(* Logix 5000 project; controller cal1632 1756-L62 rev 16.20; software revision 16.05; part 31 of 61 *)
(* tags used below, declared in another part *)
   FAULT : BOOL;
   p01r09_pb_global_reset : BOOL;
   p21_ai_splice_platen_temp : REAL;
   p21_ao_splice_platen_temp_cv : REAL;
   p21_di_close_exit_clamp : BOOL;
   p21_di_close_inlet_clamp : BOOL;
   p21_di_open_splice_platen : BOOL;
   p21_di_platen_hi_temp_ok : BOOL;
   p21_di_platen_not_closed : BOOL;
   p21_di_splice_2_hand_close : BOOL;
   p21_di_tc_bo : BOOL;
   p21_dint_to_hmi : DINT[16];
   p21_do_close_exit_clamp_sv : BOOL;
   p21_do_close_inlet_clamp_sv : BOOL;
   p21_do_close_platen_sv : BOOL;
   p21_do_enable_platen_heater : BOOL;
   p21_real_to_hmi : REAL[112];
   p21_splice_press_temp_out : SYS_SCP;
   p21_splice_temp_in_max : REAL;
   p21_splice_temp_in_min : REAL;
   p21_splice_temp_out_max : REAL;
   p21_splice_temp_out_min : REAL;
   P21r01 : routine;
   p21r02 : routine;
   p21r02_fault_exists : BOOL;
   p21r02_timer_fault : TIMER[4];
   p21r02_timer_warning : TIMER[4];
   p21r02_unack_fault : BOOL;
   p21r02_unack_warning : BOOL;
   p21r02_warning_exists : BOOL;
   p21r03 : routine;
   p21r03_timer_fault : TIMER[4];
   p21r03_timer_warning : TIMER[4];
   p21r04 : routine;
   p21r04_timer_fault : TIMER[4];
   p21r04_timer_warning : TIMER[4];
   p21r05 : routine;
   p21r05_timer_fault : TIMER[4];
   p21r05_timer_warning : TIMER[4];
   p21r06 : routine;
   p21r06_timer_fault : TIMER[4];
   p21r06_timer_warning : TIMER[4];
   p21r07 : routine;
   p21r08 : routine;
   p21r09 : routine;
   p21r10 : routine;
   p21r10_remaining_cure_time_sec : REAL;
   p21r10_status : DINT;
   p21r16 : routine;
   p21r16_pid_temp_cv : REAL;
   p21r16_request_heat : BOOL;

PROGRAM P21_Splice_Press   (* main routine R01_Main *)

ROUTINE R01_Main   (* ladder *)
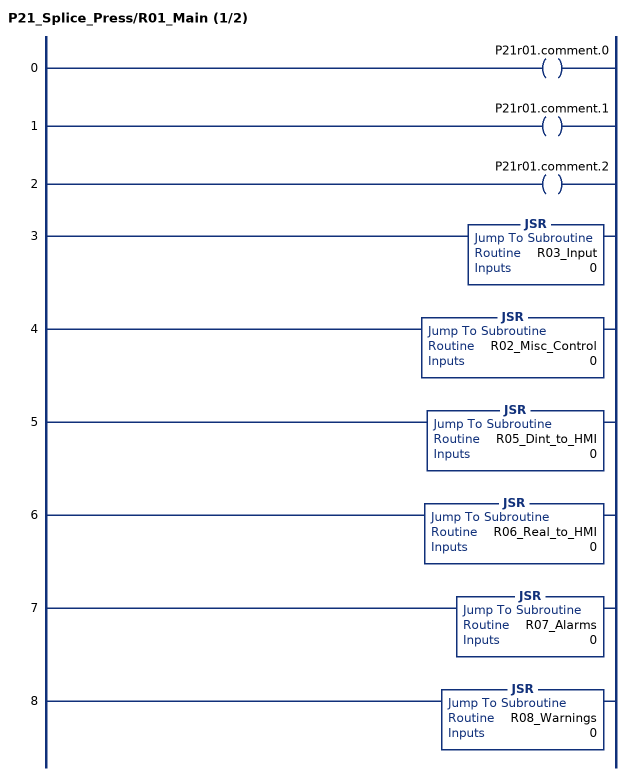
   0: OTE(P21r01.comment.0);
   1: OTE(P21r01.comment.1);
   2: OTE(P21r01.comment.2);
   3: JSR(R03_Input,0);
   4: JSR(R02_Misc_Control,0);
   5: JSR(R05_Dint_to_HMI,0);
   6: JSR(R06_Real_to_HMI,0);
   7: JSR(R07_Alarms,0);
   8: JSR(R08_Warnings,0);
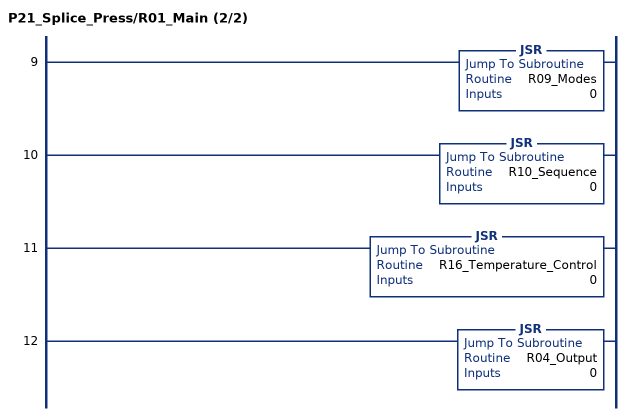
   9: JSR(R09_Modes,0);
   10: JSR(R10_Sequence,0);
   11: JSR(R16_Temperature_Control,0);
   12: JSR(R04_Output,0);
END_ROUTINE

ROUTINE R02_Misc_Control   (* ladder *)
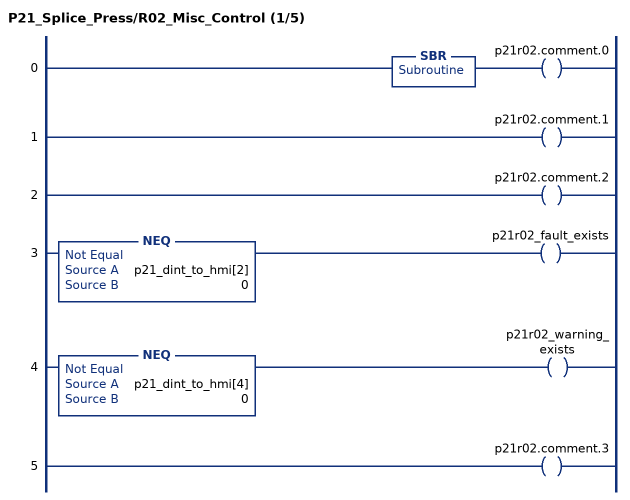
   0: SBR()OTE(p21r02.comment.0);
   1: OTE(p21r02.comment.1);
   2: OTE(p21r02.comment.2);
   3: NEQ(p21_dint_to_hmi[2],0)OTE(p21r02_fault_exists);
   4: NEQ(p21_dint_to_hmi[4],0)OTE(p21r02_warning_exists);
   5: OTE(p21r02.comment.3);
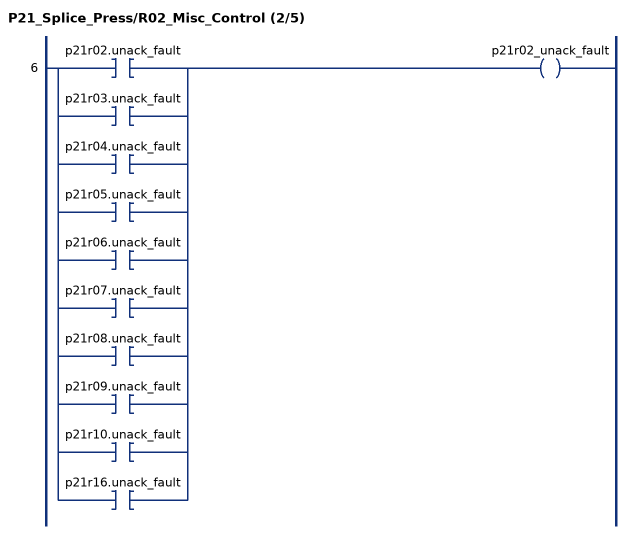
   6: [XIC(p21r02.unack_fault) ,XIC(p21r03.unack_fault) ,XIC(p21r04.unack_fault) ,XIC(p21r05.unack_fault) ,XIC(p21r06.unack_fault) ,XIC(p21r07.unack_fault) ,XIC(p21r08.unack_fault) ,XIC(p21r09.unack_fault) ,XIC(p21r10.unack_fault) ,XIC(p21r16.unack_fault) ]OTE(p21r02_unack_fault);
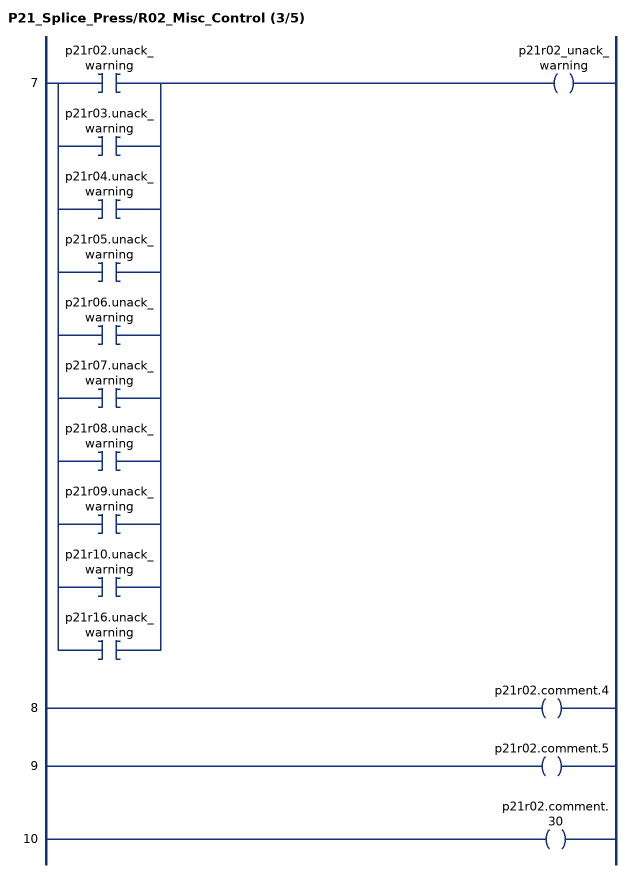
   7: [XIC(p21r02.unack_warning) ,XIC(p21r03.unack_warning) ,XIC(p21r04.unack_warning) ,XIC(p21r05.unack_warning) ,XIC(p21r06.unack_warning) ,XIC(p21r07.unack_warning) ,XIC(p21r08.unack_warning) ,XIC(p21r09.unack_warning) ,XIC(p21r10.unack_warning) ,XIC(p21r16.unack_warning) ]OTE(p21r02_unack_warning);
   8: OTE(p21r02.comment.4);
   9: OTE(p21r02.comment.5);
   10: OTE(p21r02.comment.30);
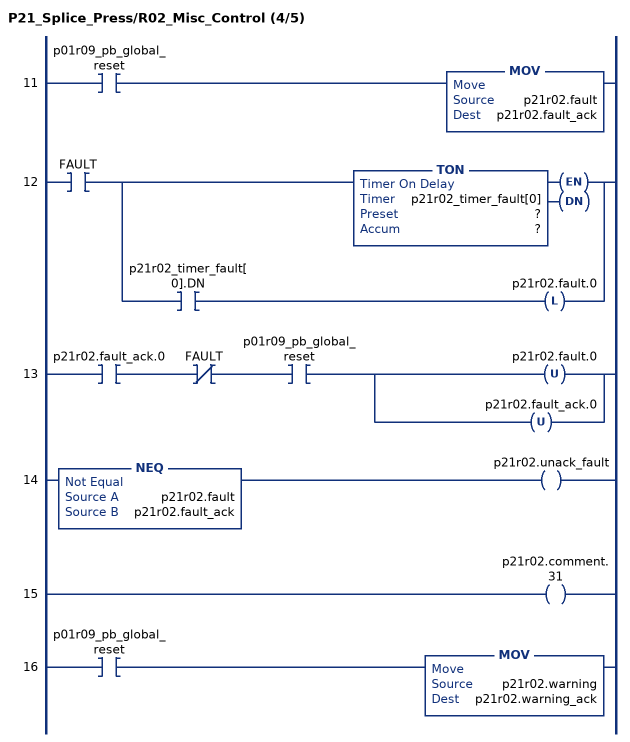
   11: XIC(p01r09_pb_global_reset)MOV(p21r02.fault,p21r02.fault_ack);
   12: XIC(FAULT)[TON(p21r02_timer_fault[0],?,?) ,XIC(p21r02_timer_fault[0].DN) OTL(p21r02.fault.0) ];
   13: XIC(p21r02.fault_ack.0)XIO(FAULT)XIC(p01r09_pb_global_reset)[OTU(p21r02.fault.0) ,OTU(p21r02.fault_ack.0) ];
   14: NEQ(p21r02.fault,p21r02.fault_ack)OTE(p21r02.unack_fault);
   15: OTE(p21r02.comment.31);
   16: XIC(p01r09_pb_global_reset)MOV(p21r02.warning,p21r02.warning_ack);
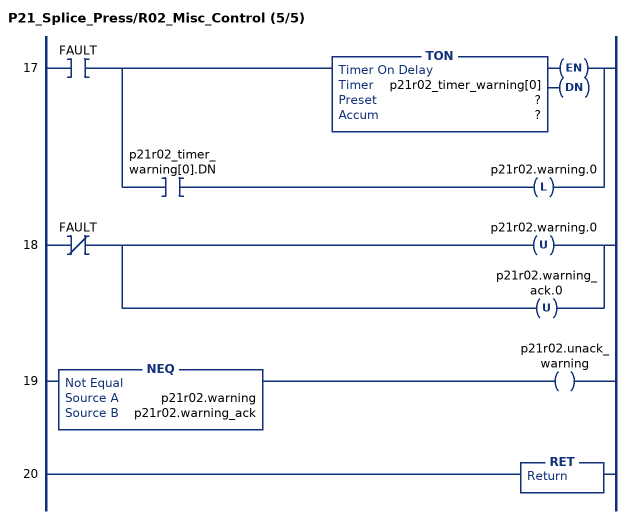
   17: XIC(FAULT)[TON(p21r02_timer_warning[0],?,?) ,XIC(p21r02_timer_warning[0].DN) OTL(p21r02.warning.0) ];
   18: XIO(FAULT)[OTU(p21r02.warning.0) ,OTU(p21r02.warning_ack.0) ];
   19: NEQ(p21r02.warning,p21r02.warning_ack)OTE(p21r02.unack_warning);
   20: RET();
END_ROUTINE

ROUTINE R03_Input   (* ladder *)
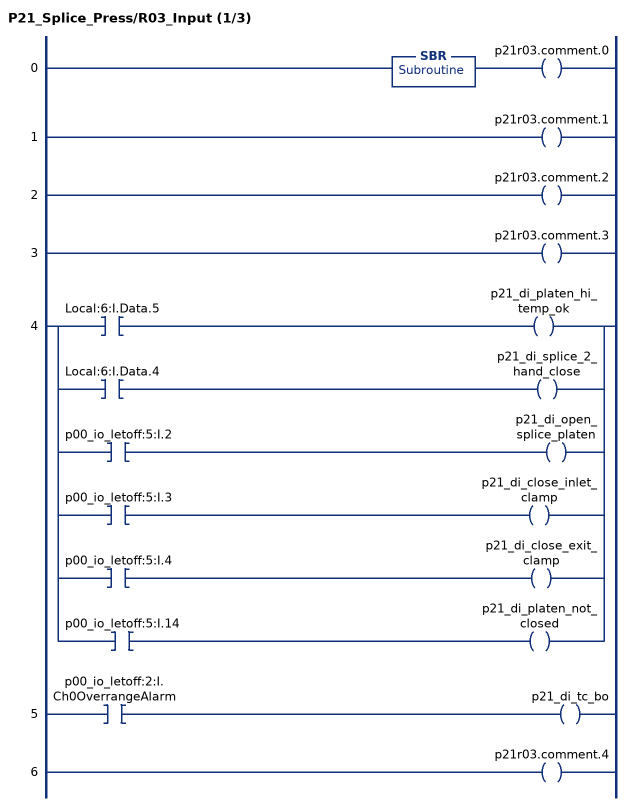
   0: SBR()OTE(p21r03.comment.0);
   1: OTE(p21r03.comment.1);
   2: OTE(p21r03.comment.2);
   3: OTE(p21r03.comment.3);
   4: [XIC(Local:6:I.Data.5) OTE(p21_di_platen_hi_temp_ok) ,XIC(Local:6:I.Data.4) OTE(p21_di_splice_2_hand_close) ,XIC(p00_io_letoff:5:I.2) OTE(p21_di_open_splice_platen) ,XIC(p00_io_letoff:5:I.3) OTE(p21_di_close_inlet_clamp) ,XIC(p00_io_letoff:5:I.4) OTE(p21_di_close_exit_clamp) ,XIC(p00_io_letoff:5:I.14) OTE(p21_di_platen_not_closed) ];
   5: XIC(p00_io_letoff:2:I.Ch0OverrangeAlarm)OTE(p21_di_tc_bo);
   6: OTE(p21r03.comment.4);
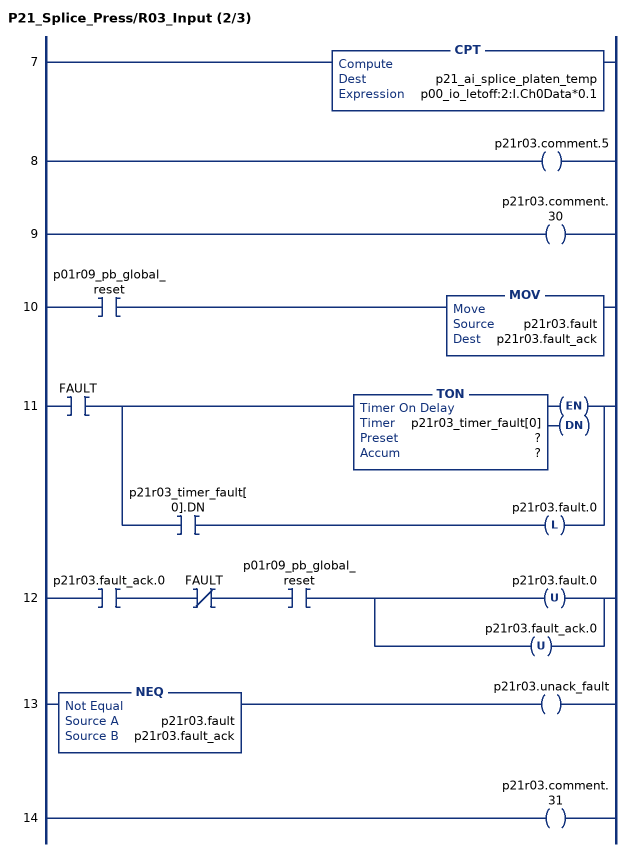
   7: CPT(p21_ai_splice_platen_temp,p00_io_letoff:2:I.Ch0Data*0.1);
   8: OTE(p21r03.comment.5);
   9: OTE(p21r03.comment.30);
   10: XIC(p01r09_pb_global_reset)MOV(p21r03.fault,p21r03.fault_ack);
   11: XIC(FAULT)[TON(p21r03_timer_fault[0],?,?) ,XIC(p21r03_timer_fault[0].DN) OTL(p21r03.fault.0) ];
   12: XIC(p21r03.fault_ack.0)XIO(FAULT)XIC(p01r09_pb_global_reset)[OTU(p21r03.fault.0) ,OTU(p21r03.fault_ack.0) ];
   13: NEQ(p21r03.fault,p21r03.fault_ack)OTE(p21r03.unack_fault);
   14: OTE(p21r03.comment.31);
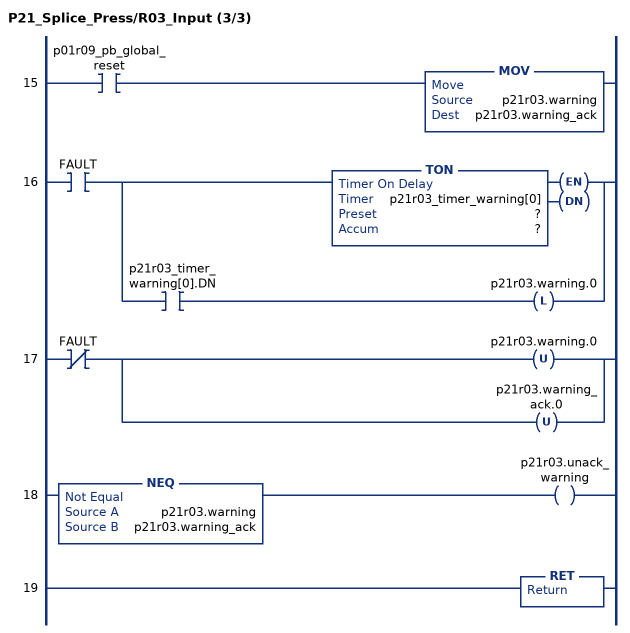
   15: XIC(p01r09_pb_global_reset)MOV(p21r03.warning,p21r03.warning_ack);
   16: XIC(FAULT)[TON(p21r03_timer_warning[0],?,?) ,XIC(p21r03_timer_warning[0].DN) OTL(p21r03.warning.0) ];
   17: XIO(FAULT)[OTU(p21r03.warning.0) ,OTU(p21r03.warning_ack.0) ];
   18: NEQ(p21r03.warning,p21r03.warning_ack)OTE(p21r03.unack_warning);
   19: RET();
END_ROUTINE

ROUTINE R04_Output   (* ladder *)
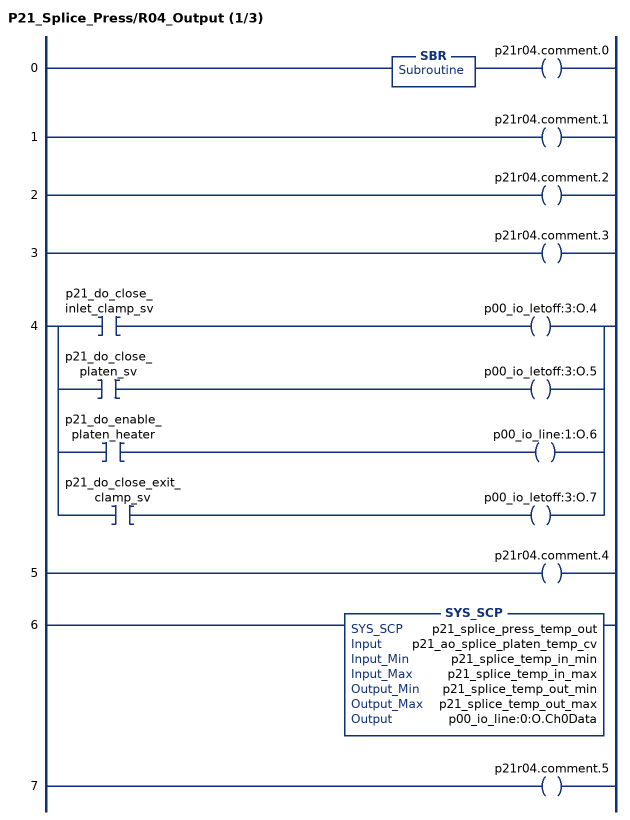
   0: SBR()OTE(p21r04.comment.0);
   1: OTE(p21r04.comment.1);
   2: OTE(p21r04.comment.2);
   3: OTE(p21r04.comment.3);
   4: [XIC(p21_do_close_inlet_clamp_sv) OTE(p00_io_letoff:3:O.4) ,XIC(p21_do_close_platen_sv) OTE(p00_io_letoff:3:O.5) ,XIC(p21_do_enable_platen_heater) OTE(p00_io_line:1:O.6) ,XIC(p21_do_close_exit_clamp_sv) OTE(p00_io_letoff:3:O.7) ];
   5: OTE(p21r04.comment.4);
   6: SYS_SCP(p21_splice_press_temp_out,p21_ao_splice_platen_temp_cv,p21_splice_temp_in_min,p21_splice_temp_in_max,p21_splice_temp_out_min,p21_splice_temp_out_max,p00_io_line:0:O.Ch0Data);
   7: OTE(p21r04.comment.5);
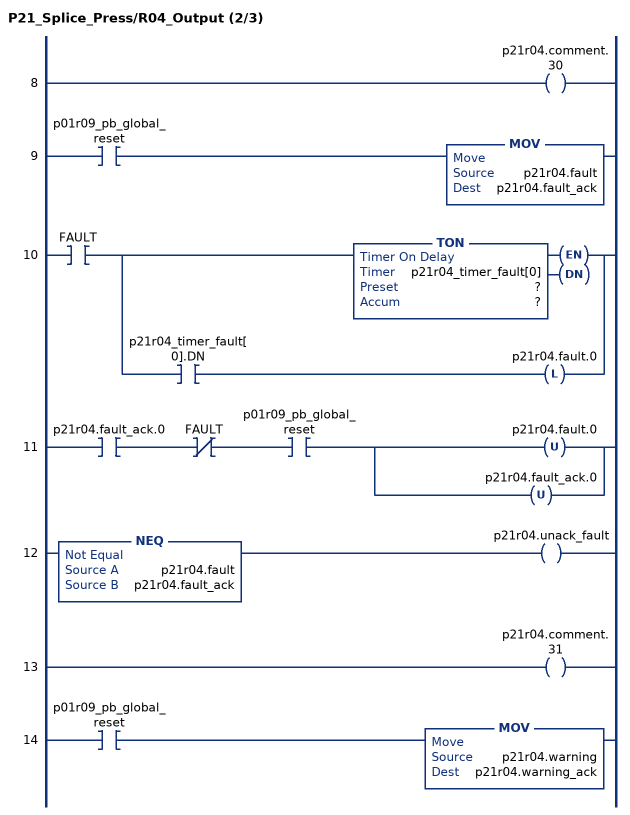
   8: OTE(p21r04.comment.30);
   9: XIC(p01r09_pb_global_reset)MOV(p21r04.fault,p21r04.fault_ack);
   10: XIC(FAULT)[TON(p21r04_timer_fault[0],?,?) ,XIC(p21r04_timer_fault[0].DN) OTL(p21r04.fault.0) ];
   11: XIC(p21r04.fault_ack.0)XIO(FAULT)XIC(p01r09_pb_global_reset)[OTU(p21r04.fault.0) ,OTU(p21r04.fault_ack.0) ];
   12: NEQ(p21r04.fault,p21r04.fault_ack)OTE(p21r04.unack_fault);
   13: OTE(p21r04.comment.31);
   14: XIC(p01r09_pb_global_reset)MOV(p21r04.warning,p21r04.warning_ack);
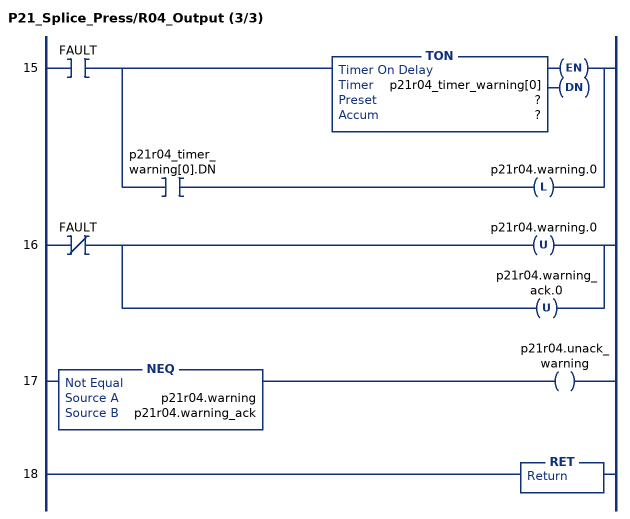
   15: XIC(FAULT)[TON(p21r04_timer_warning[0],?,?) ,XIC(p21r04_timer_warning[0].DN) OTL(p21r04.warning.0) ];
   16: XIO(FAULT)[OTU(p21r04.warning.0) ,OTU(p21r04.warning_ack.0) ];
   17: NEQ(p21r04.warning,p21r04.warning_ack)OTE(p21r04.unack_warning);
   18: RET();
END_ROUTINE

ROUTINE R05_Dint_to_HMI   (* ladder *)
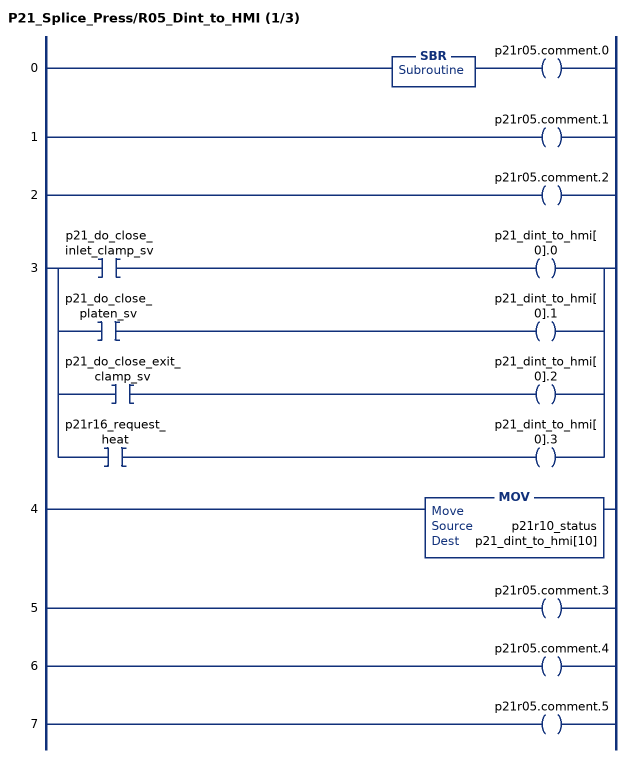
   0: SBR()OTE(p21r05.comment.0);
   1: OTE(p21r05.comment.1);
   2: OTE(p21r05.comment.2);
   3: [XIC(p21_do_close_inlet_clamp_sv) OTE(p21_dint_to_hmi[0].0) ,XIC(p21_do_close_platen_sv) OTE(p21_dint_to_hmi[0].1) ,XIC(p21_do_close_exit_clamp_sv) OTE(p21_dint_to_hmi[0].2) ,XIC(p21r16_request_heat) OTE(p21_dint_to_hmi[0].3) ];
   4: MOV(p21r10_status,p21_dint_to_hmi[10]);
   5: OTE(p21r05.comment.3);
   6: OTE(p21r05.comment.4);
   7: OTE(p21r05.comment.5);
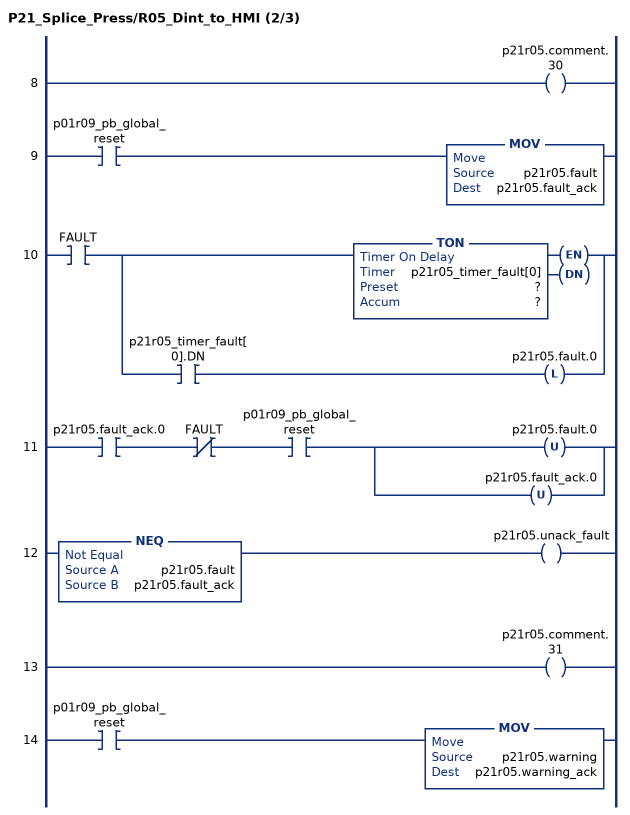
   8: OTE(p21r05.comment.30);
   9: XIC(p01r09_pb_global_reset)MOV(p21r05.fault,p21r05.fault_ack);
   10: XIC(FAULT)[TON(p21r05_timer_fault[0],?,?) ,XIC(p21r05_timer_fault[0].DN) OTL(p21r05.fault.0) ];
   11: XIC(p21r05.fault_ack.0)XIO(FAULT)XIC(p01r09_pb_global_reset)[OTU(p21r05.fault.0) ,OTU(p21r05.fault_ack.0) ];
   12: NEQ(p21r05.fault,p21r05.fault_ack)OTE(p21r05.unack_fault);
   13: OTE(p21r05.comment.31);
   14: XIC(p01r09_pb_global_reset)MOV(p21r05.warning,p21r05.warning_ack);
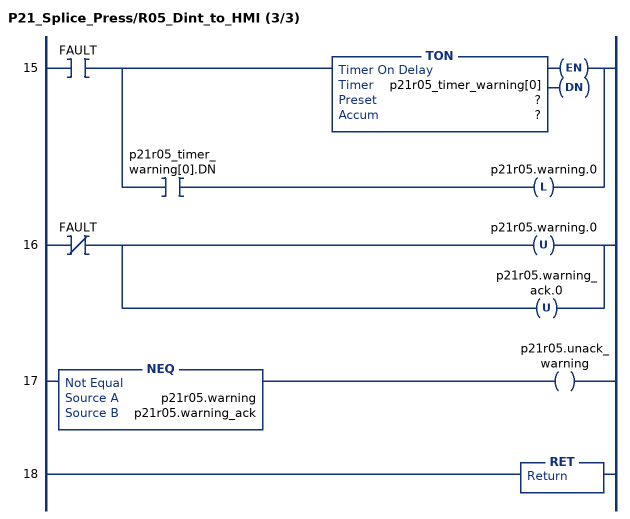
   15: XIC(FAULT)[TON(p21r05_timer_warning[0],?,?) ,XIC(p21r05_timer_warning[0].DN) OTL(p21r05.warning.0) ];
   16: XIO(FAULT)[OTU(p21r05.warning.0) ,OTU(p21r05.warning_ack.0) ];
   17: NEQ(p21r05.warning,p21r05.warning_ack)OTE(p21r05.unack_warning);
   18: RET();
END_ROUTINE

ROUTINE R06_Real_to_HMI   (* ladder *)
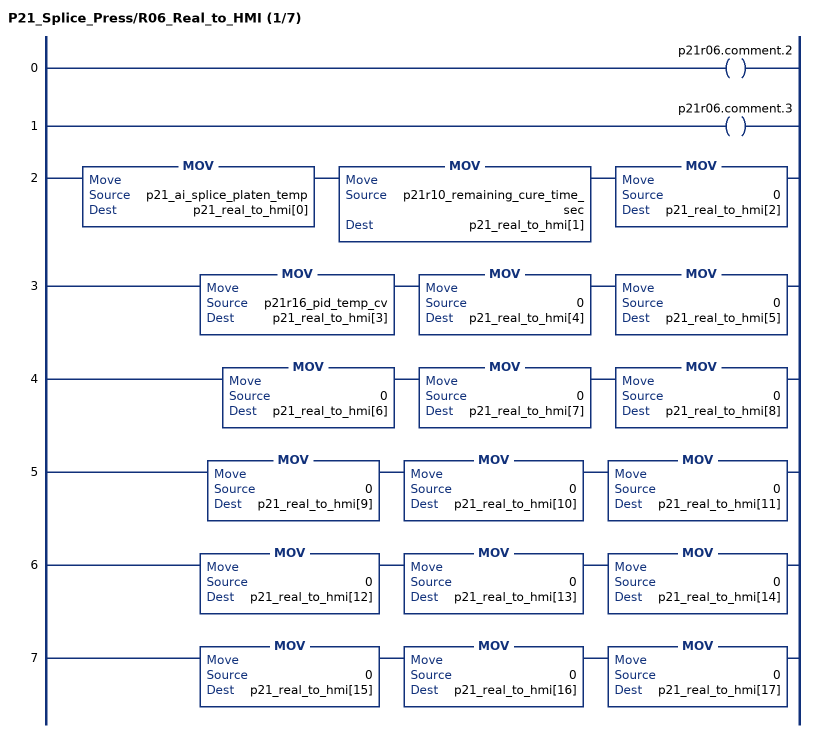
   0: OTE(p21r06.comment.2);
   1: OTE(p21r06.comment.3);
   2: MOV(p21_ai_splice_platen_temp,p21_real_to_hmi[0])MOV(p21r10_remaining_cure_time_sec,p21_real_to_hmi[1])MOV(0,p21_real_to_hmi[2]);
   3: MOV(p21r16_pid_temp_cv,p21_real_to_hmi[3])MOV(0,p21_real_to_hmi[4])MOV(0,p21_real_to_hmi[5]);
   4: MOV(0,p21_real_to_hmi[6])MOV(0,p21_real_to_hmi[7])MOV(0,p21_real_to_hmi[8]);
   5: MOV(0,p21_real_to_hmi[9])MOV(0,p21_real_to_hmi[10])MOV(0,p21_real_to_hmi[11]);
   6: MOV(0,p21_real_to_hmi[12])MOV(0,p21_real_to_hmi[13])MOV(0,p21_real_to_hmi[14]);
   7: MOV(0,p21_real_to_hmi[15])MOV(0,p21_real_to_hmi[16])MOV(0,p21_real_to_hmi[17]);
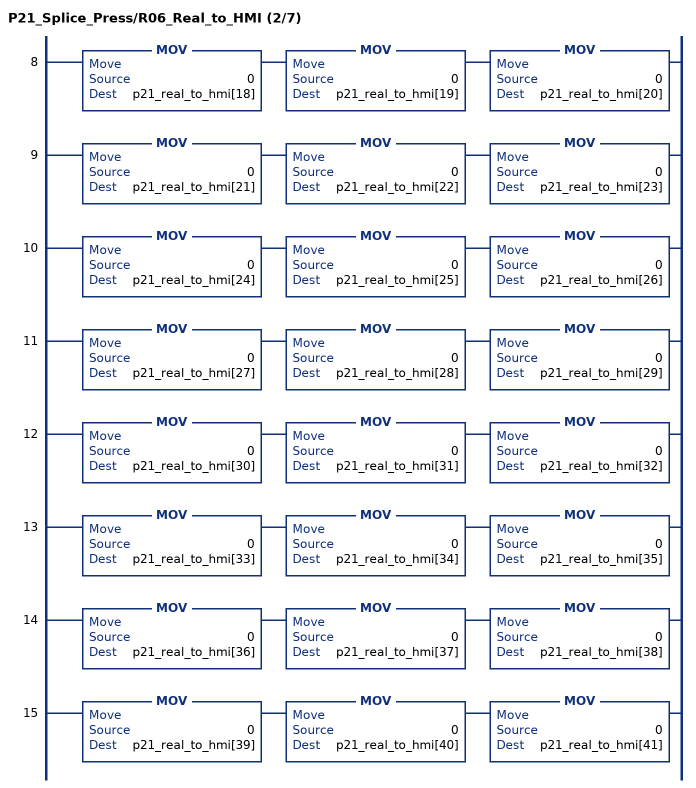
   8: MOV(0,p21_real_to_hmi[18])MOV(0,p21_real_to_hmi[19])MOV(0,p21_real_to_hmi[20]);
   9: MOV(0,p21_real_to_hmi[21])MOV(0,p21_real_to_hmi[22])MOV(0,p21_real_to_hmi[23]);
   10: MOV(0,p21_real_to_hmi[24])MOV(0,p21_real_to_hmi[25])MOV(0,p21_real_to_hmi[26]);
   11: MOV(0,p21_real_to_hmi[27])MOV(0,p21_real_to_hmi[28])MOV(0,p21_real_to_hmi[29]);
   12: MOV(0,p21_real_to_hmi[30])MOV(0,p21_real_to_hmi[31])MOV(0,p21_real_to_hmi[32]);
   13: MOV(0,p21_real_to_hmi[33])MOV(0,p21_real_to_hmi[34])MOV(0,p21_real_to_hmi[35]);
   14: MOV(0,p21_real_to_hmi[36])MOV(0,p21_real_to_hmi[37])MOV(0,p21_real_to_hmi[38]);
   15: MOV(0,p21_real_to_hmi[39])MOV(0,p21_real_to_hmi[40])MOV(0,p21_real_to_hmi[41]);
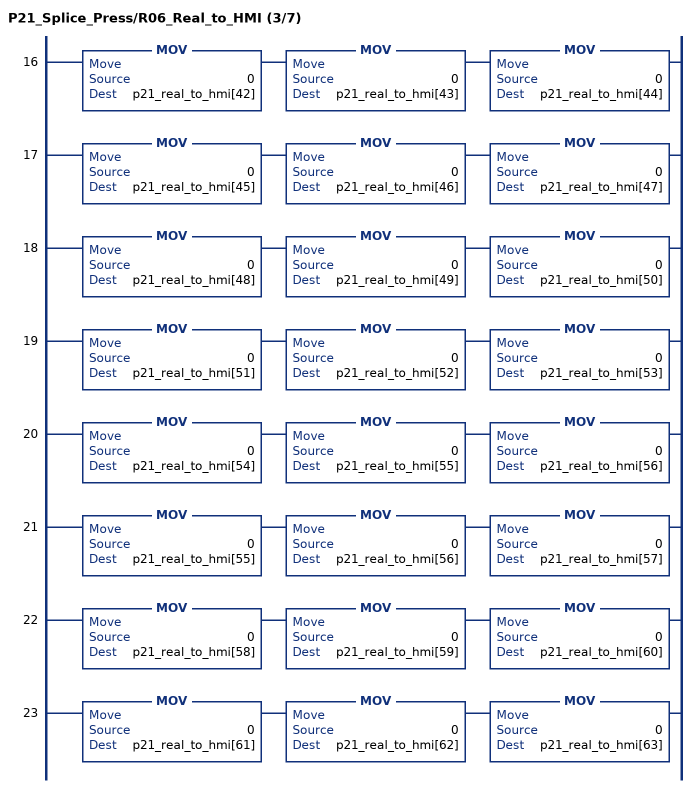
   16: MOV(0,p21_real_to_hmi[42])MOV(0,p21_real_to_hmi[43])MOV(0,p21_real_to_hmi[44]);
   17: MOV(0,p21_real_to_hmi[45])MOV(0,p21_real_to_hmi[46])MOV(0,p21_real_to_hmi[47]);
   18: MOV(0,p21_real_to_hmi[48])MOV(0,p21_real_to_hmi[49])MOV(0,p21_real_to_hmi[50]);
   19: MOV(0,p21_real_to_hmi[51])MOV(0,p21_real_to_hmi[52])MOV(0,p21_real_to_hmi[53]);
   20: MOV(0,p21_real_to_hmi[54])MOV(0,p21_real_to_hmi[55])MOV(0,p21_real_to_hmi[56]);
   21: MOV(0,p21_real_to_hmi[55])MOV(0,p21_real_to_hmi[56])MOV(0,p21_real_to_hmi[57]);
   22: MOV(0,p21_real_to_hmi[58])MOV(0,p21_real_to_hmi[59])MOV(0,p21_real_to_hmi[60]);
   23: MOV(0,p21_real_to_hmi[61])MOV(0,p21_real_to_hmi[62])MOV(0,p21_real_to_hmi[63]);
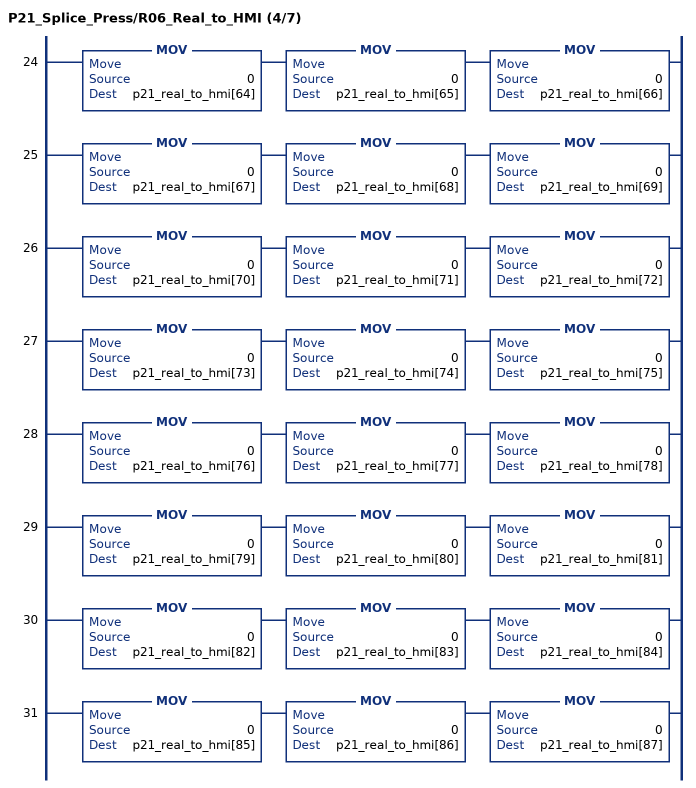
   24: MOV(0,p21_real_to_hmi[64])MOV(0,p21_real_to_hmi[65])MOV(0,p21_real_to_hmi[66]);
   25: MOV(0,p21_real_to_hmi[67])MOV(0,p21_real_to_hmi[68])MOV(0,p21_real_to_hmi[69]);
   26: MOV(0,p21_real_to_hmi[70])MOV(0,p21_real_to_hmi[71])MOV(0,p21_real_to_hmi[72]);
   27: MOV(0,p21_real_to_hmi[73])MOV(0,p21_real_to_hmi[74])MOV(0,p21_real_to_hmi[75]);
   28: MOV(0,p21_real_to_hmi[76])MOV(0,p21_real_to_hmi[77])MOV(0,p21_real_to_hmi[78]);
   29: MOV(0,p21_real_to_hmi[79])MOV(0,p21_real_to_hmi[80])MOV(0,p21_real_to_hmi[81]);
   30: MOV(0,p21_real_to_hmi[82])MOV(0,p21_real_to_hmi[83])MOV(0,p21_real_to_hmi[84]);
   31: MOV(0,p21_real_to_hmi[85])MOV(0,p21_real_to_hmi[86])MOV(0,p21_real_to_hmi[87]);
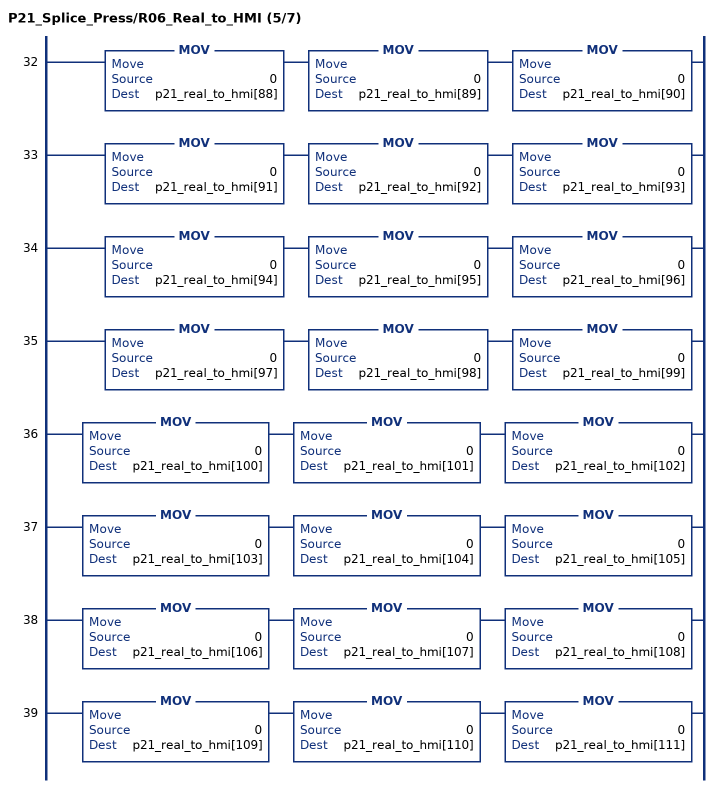
   32: MOV(0,p21_real_to_hmi[88])MOV(0,p21_real_to_hmi[89])MOV(0,p21_real_to_hmi[90]);
   33: MOV(0,p21_real_to_hmi[91])MOV(0,p21_real_to_hmi[92])MOV(0,p21_real_to_hmi[93]);
   34: MOV(0,p21_real_to_hmi[94])MOV(0,p21_real_to_hmi[95])MOV(0,p21_real_to_hmi[96]);
   35: MOV(0,p21_real_to_hmi[97])MOV(0,p21_real_to_hmi[98])MOV(0,p21_real_to_hmi[99]);
   36: MOV(0,p21_real_to_hmi[100])MOV(0,p21_real_to_hmi[101])MOV(0,p21_real_to_hmi[102]);
   37: MOV(0,p21_real_to_hmi[103])MOV(0,p21_real_to_hmi[104])MOV(0,p21_real_to_hmi[105]);
   38: MOV(0,p21_real_to_hmi[106])MOV(0,p21_real_to_hmi[107])MOV(0,p21_real_to_hmi[108]);
   39: MOV(0,p21_real_to_hmi[109])MOV(0,p21_real_to_hmi[110])MOV(0,p21_real_to_hmi[111]);
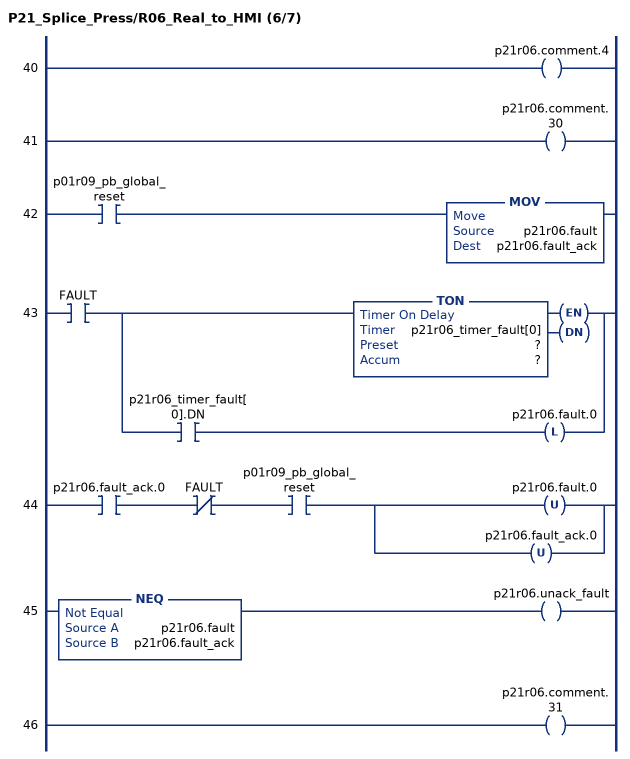
   40: OTE(p21r06.comment.4);
   41: OTE(p21r06.comment.30);
   42: XIC(p01r09_pb_global_reset)MOV(p21r06.fault,p21r06.fault_ack);
   43: XIC(FAULT)[TON(p21r06_timer_fault[0],?,?) ,XIC(p21r06_timer_fault[0].DN) OTL(p21r06.fault.0) ];
   44: XIC(p21r06.fault_ack.0)XIO(FAULT)XIC(p01r09_pb_global_reset)[OTU(p21r06.fault.0) ,OTU(p21r06.fault_ack.0) ];
   45: NEQ(p21r06.fault,p21r06.fault_ack)OTE(p21r06.unack_fault);
   46: OTE(p21r06.comment.31);
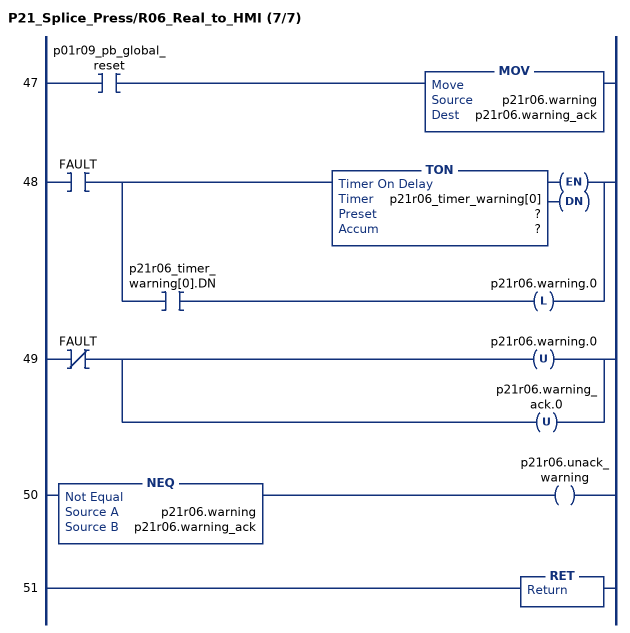
   47: XIC(p01r09_pb_global_reset)MOV(p21r06.warning,p21r06.warning_ack);
   48: XIC(FAULT)[TON(p21r06_timer_warning[0],?,?) ,XIC(p21r06_timer_warning[0].DN) OTL(p21r06.warning.0) ];
   49: XIO(FAULT)[OTU(p21r06.warning.0) ,OTU(p21r06.warning_ack.0) ];
   50: NEQ(p21r06.warning,p21r06.warning_ack)OTE(p21r06.unack_warning);
   51: RET();
END_ROUTINE
